{attribute addProperty BoxType "EM7004-0000-0017"}
{attribute addProperty Id "PLS_EnabledBIT10.1251Unequal_SI_0BIT10.1252"}
{attribute addProperty CRC "3419751092"}
{attribute addProperty SizeInBites "16"}
{attribute addProperty SizeInBytes "2"}
TYPE Status_CBD542B4 :
STRUCT
	{attribute addProperty Name "PLS_Enabled"}
	PLS_Enabled : BIT;
	{attribute addProperty Name "Unequal_SI_0"}
	Unequal_SI_0 : BIT;
	{attribute 'hide'}
	reserve_1_BIT_0 : BIT;
	{attribute 'hide'}
	reserve_1_BIT_1 : BIT;
	{attribute 'hide'}
	reserve_1_BIT_2 : BIT;
	{attribute 'hide'}
	reserve_1_BIT_3 : BIT;
	{attribute 'hide'}
	reserve_1_BIT_4 : BIT;
	{attribute 'hide'}
	reserve_1_BIT_5 : BIT;
	{attribute 'hide'}
	reserve_1_BIT_6 : BIT;
	{attribute 'hide'}
	reserve_1_BIT_7 : BIT;
	{attribute 'hide'}
	reserve_1_BIT_8 : BIT;
	{attribute 'hide'}
	reserve_1_BIT_9 : BIT;
	{attribute 'hide'}
	reserve_1_BIT_10 : BIT;
	{attribute 'hide'}
	reserve_1_BIT_11 : BIT;
	{attribute 'hide'}
	reserve_1_BIT_12 : BIT;
	{attribute 'hide'}
	reserve_1_BIT_13 : BIT;
END_STRUCT
END_TYPE

(* stored: Version 1.2.0.0, ProductVersion 3.1.4024.9
   DUT Status_CBD542B4: Id {087d1893-eb4b-4347-972a-ad8f86e157ef} *)
